PROGRAM MAIN
VAR
END_VAR

END_PROGRAM

(* stored: Version 1.1.0.1
   POU MAIN: Id {55dc8056-a83c-498b-9d09-689d30efbd92} *)
